// TIA Portal V16 export
// export: Created 2023-09-11T12:14:55.7817244Z, ExportSetting WithDefaults, DisplayName Totally Integrated Automation Portal, DisplayVersion V16 Update 6, DisplayName TIA Portal Version Control Interface, DisplayVersion V16 Update 2, DisplayName TIA Portal Openness, DisplayVersion V16 Update 6, DisplayName STEP 7 Professional, DisplayVersion V16 Update 6, DisplayName STEP 7 Safety, DisplayVersion V16, DisplayName WinCC Advanced, DisplayVersion V16 Update 6
DATA_BLOCK "dbHoldRegSlave_to_MT101"   // DB100
{ S7_Optimized_Access := 'FALSE' }
VERSION : 0.1
// stored: AutoNumber false, DBAccessibleFromOPCUA true, IsOnlyStoredInLoadMemory false, IsWriteProtectedInAS false
   VAR
      instPump1 : Word := 33924;   // 40001 Pompa Status M1
      instPump2 : Word := 33924;   // 40002 Pompa Status M2
      instPump3 : Word := 33924;   // 40003 Pompa Status M3
      instPump4 : Word := 33924;   // 40004 Pompa Status M4
      instvValveZ1 : Word := 0;   // 40005 Zasuwa Status Z1
      instvValveZ2 : Word := 0;   // 40006 Zasuwa Status Z2
      instvValveZ3 : Word := 0;   // 40007 Zasuwa Status Z3
      instvValveZ4 : Word := 0;   // 40008 Zasuwa Status Z4
      instvValveZ5 : Word := 0;   // 40009 Zasuwa Status Z5
      instvValveZ6 : Word := 0;   // 40010 Zasuwa Status Z6
      instvValveZ7 : Word := 0;   // 40011 Zasuwa Status Z7
      instvValveZ8 : Word := 0;   // 40012 Zasuwa Status Z8
      instvValveZ9 : Word := 0;   // 40013 Zasuwa Status Z9
      instvValveZ10 : Word := 0;   // 40014 Zasuwa Status Z10
      instvValveZ11 : Word := 33924;   // 40015 Zasuwa Status Z11
      instvValveZ12 : Word := 0;   // 40016 Zasuwa Status Z12
      instControllDrivers_1 : Int := 0;   // Bity sterowania napędami (start, stop, otwórz, zamknij) / 40017 Bity sterowania napędami (start, stop, otwórz, zamknij) Pompami M1-M4, Zasuwami Z1, Z2, Z3, Z4
      instControllDrivers_2 : Int := 0;   // Bity przełączenia trybu pracy napędów / 40018 Bity sterowania napędami ( otwórz, zamknij, start, stop) Zasuwami Z5, Z6, Z7, Z8, Z9, Z10, Z11, Z12
      instConrol_ManAut_1 : Int := 0;   // Bity przełączenia trybu pracy napędów / 40019 Bity przełączenia trybu pracy napędów M1-M4, Zasuwami Z1, Z2, Z3, Z4
      instConrol_ManAut_2 : Int := 0;   // Bity przełączenia trybu pracy napędów / 40020 Bity przełączenia trybu pracy napędów Z5, Z6, Z7, Z8, Z9, Z10, Z11, Z12
      instLevelTank1 : Int := 0;   // Poziom zbiornik / 40021 Poziom zbiornik
      instLevelTank2 : Int := 0;   // Poziom zbiornik / 40022 Poziom zbiornik
      instLevelTank3 : Int := 0;   // Poziom zbiornik / 40023 Poziom zbiornik
      instLevelTank4 : Int := 0;   // Poziom zbiornik / 40024 Poziom zbiornik
      instPosition_Z10 : Int;   // rezerwa / 40025 Zadawanie położenia Z10
      instClearFault1 : Int := 0;   // Bity kasowania alarmów napędów M1-M4, Z1 - Z12 / 40026 Bity kasowania alarmów napędów M1-M4, Z1 - Z12
      instSygSter_1 : Int;   // rezerwa / 40027 Sygnały sterowania strategią pompownia - 0= wyłaczone, 1=dosilanie, 2=przetłaczanie,3=automat, 4=ręczne
      instSygSter_2 : Int;   // 40028 Sygnały sterowania cyklem zbiorniki 0-wyłączone, 1=dobowy, 2=sekwencyjny, 3=ręczne
      instCurrent_Inverter : Int := 0;   // 40029 Aktualny prądu falownika
      instHz_Inverter : Int := 0;   // 40030 Aktualne Hz na falowniku
      instLevelSetFilling : Real;   // 40031 Zadany poziom napełniania
      instLevelSetEmptying : Real;   // 40033 Zadany poziom opróżniania
      instSetbarDN225_B6 : Real;   // 40035 Zadany ciśnienie tłóczenia kierunek miasto, Modbus 40035
      instSetbarDN500_B5 : Real;   // 40037 Zadana ciśnienie dosilania kierunek dosilanie "0" Modbus 40037
      instSetBarMinB9 : Real;   // 40039 Zadawana dolna granica ciśnienia magistrala C1 Wielkopolska 40039
      instB5bar_act : Real;   // 40041 Aktualne ciśnienie zasilania z sieci
      instB6bar_act : Real;   // 40043 Aktualne ciśnienie DN225 tłoczny
      instB7bar_act : Real;   // 40045 Aktualne ciśnienie DN225 pompy
      instB8bar_act : Real;   // 40047 Aktualne ciśnienie ssoncy pomp (zab. Suchobieg)
      instPozitionZ10_act : Real;   // 40049 Aktualna pozycja zasuwy Z10
      instFlowDN225_act : Real;   // 40051 Przepływ DN225 aktualny MIASTO
      instFlowDN225_sum : Real;   // 40053 SUMA przepływu Dolna DN225
      instFlowDN500_act : Real;   // 40055 Przepływ DN500 (l/s) aktualny, zasilanie zbiorników, DOSILANIE, Modbus 40055
      instFlowDN500_sum : Real;   // 40057 SUMA przepływu Dolna DN500 Modbus 40057
      instHourStart_Filling : Int;   // 40059 Godzina start napełniania
      instMinutStart_Filling : Int;   // 40060 Minuta start napełniania
      instHourStop_Filling : Int;   // 40061 Godzina stop napełniania
      instMinutStopt_Filling : Int;   // 40062 Minuta stop napełniania
      instHourStart_City : Int;   // 40063 Godzina start przetłaczanie miasto DN225
      instMinutStart_City : Int;   // 40064 Minuty start przetłaczanie miasto DN225
      instHourStop_City : Int;   // 40065 Godzina stop przetłaczanie miasto DN225
      instMinutStopt_City : Int;   // 40066 Minuty stop przetłaczanie miasto DN225
      instHourStart_Replen : Int;   // 40067 Godzina start przetłaczanie magistrala DN500
      instMinutStart_Replen : Int;   // 40068 Minuty start przetłaczanie magistrala DN500
      instHourStop_Replen : Int;   // 40069 Godzina stop przetłaczanie magistrala DN500
      instMinutStopt_Replen : Int;   // 40070 Minuty stop przetłaczanie magistrala DN500
   END_VAR
BEGIN
END_DATA_BLOCK
